// TIA Portal V20 export
ORGANIZATION_BLOCK "Startup"   // OB1030, LAD, Startup
TITLE = "Complete Restart"
AUTHOR : ERsystem_FA2_DH. Kim
// stored: AutoNumber false, IsIECCheckEnabled true, Namespace Unit1.Em3, SetENOAutomatically false
   VAR_INPUT
      LostRetentive : Bool;   // True if retentive data are lost
      LostRTC : Bool;   // True if date and time are lost
   END_VAR
BEGIN

REGION Network 1 (SCL): Build the Absolut Reference Designator
   // Set the Absoult Reference Designator in the Config DB
   IF LEN(IN := "Unit1.Em3.Config".em.referenceDesignator.parent) <> 0 THEN
     "Unit1.Em3.Config".em.referenceDesignator.combined := CONCAT_WSTRING(IN1 := "Unit1.Em3.Config".em.referenceDesignator.parent, IN2 := WSTRING#'.', IN3 := "Unit1.Em3.Config".em.referenceDesignator.relative);
   ELSE
     "Unit1.Em3.Config".em.referenceDesignator.combined := "Unit1.Em3.Config".em.referenceDesignator.relative;
   END_IF;
END_REGION

REGION Network 2 (SCL): Assign axes data
   //Assign axes
   "Unit1.Em3.Config".axis[1] := "BA030AZSDR3_CompensatorAxisX";
   // Config.axis[2] := _."BA030A_MasterAxis";
   "Unit1.Em3.Config".axis[3] := "BA030A_UnwinderVirtualAxis";

   "Unit1.Em3.Config".cam[1] := "BA030AZSDR3_CompensatorAxisXCamMain";
   "Unit1.Em3.Config".cam[2] := "BA030AZSDR3_CompensatorAxisXCamSub";

   // Assign configuration data of axis

   // FB Enable
   "Unit1.Em3.HmiInterface".cmCompensatorAxisX.commands.enableMasterControl := TRUE;
END_REGION

REGION Network 3 (SCL): Assign TwoWayActuator data
   //Assgin Configuration data of TwoWayActuator
   "Unit1.Em3.Config".cmDancerFwdBwd.disableFeedbackHomePos := TRUE;
   "Unit1.Em3.Config".cmDancerFwdBwd.disableFeedbackWorkPos := TRUE;

   "Unit1.Em3.Config".cmDancerFwdBwd.monitoringLeavingFeedback := t#1000ms;
   "Unit1.Em3.Config".cmDancerFwdBwd.monitoringReachingFeedback := t#1000ms;

   "Unit1.Em3.Config".cmSepaUnwinderIonizerTop.disableFeedbackHomePos := TRUE;
   "Unit1.Em3.Config".cmSepaUnwinderIonizerTop.disableFeedbackWorkPos := TRUE;

   "Unit1.Em3.Config".cmSepaUnwinderIonizerBottom.disableFeedbackHomePos := TRUE;
   "Unit1.Em3.Config".cmSepaUnwinderIonizerBottom.disableFeedbackWorkPos := TRUE;
END_REGION

REGION Network 4 (SCL): Assign EPC Config
   "Unit1.Em3.Config".cmEpcPivot.hwID.EkrOut_Auto_Sp_Acp_HW_ID := 1077;
   "Unit1.Em3.Config".cmEpcPivot.hwID.EkrOut_CAM_Data_HW_ID := 1078;
   "Unit1.Em3.Config".cmEpcPivot.hwID.EkrOut_CLS_Data_HW_ID := 1079;
   "Unit1.Em3.Config".cmEpcPivot.hwID.EkrOut_Guiding_edges_HW_ID := 1081;
   "Unit1.Em3.Config".cmEpcPivot.hwID.EkrOut_HEADER_Data_HW_ID := 1082;
   "Unit1.Em3.Config".cmEpcPivot.hwID.EkrOut_POS_unit_HW_ID := 1084;
   "Unit1.Em3.Config".cmEpcPivot.hwID.EkrOut_SEN_Data_HW_ID := 1085;
   "Unit1.Em3.Config".cmEpcPivot.hwID.EkrOut_Servo_Center_HW_ID := 1086;
   "Unit1.Em3.Config".cmEpcPivot.hwID.EkrOut_Setpoint_HW_ID := 1087;
   "Unit1.Em3.Config".cmEpcPivot.hwID.EkrOut_Web_width_HW_ID := 1088;
   "Unit1.Em3.Config".cmEpcPivot.hwID.EkrIn_Auto_Sp_Acp_HW_ID := 1089;
   "Unit1.Em3.Config".cmEpcPivot.hwID.EkrIn_HEADER_Data_HW_ID := 1091;
   "Unit1.Em3.Config".cmEpcPivot.hwID.EkrIn_POS_unit_HW_ID := 1093;
   "Unit1.Em3.Config".cmEpcPivot.hwID.EkrIn_Setpoint_HW_ID := 1094;
   "Unit1.Em3.Config".cmEpcPivot.hwID.EkrIn_Web_width_HW_ID := 1095;
END_REGION
END_ORGANIZATION_BLOCK
